FUNCTION DT_TO_SDT : SDT
VAR_INPUT
	DTI : DT;
END_VAR
VAR
	tmp : DATE;
	tdt : DWORD;
END_VAR


(*
version 1.0	18. oct 2008
programmer 	hugo
tested by	oscat

converts date_time to Structured date time (SDT)

*)

tmp := DT_TO_DATE(dti);
tdt := DT_TO_DWORD(dti) - DATE_TO_DWORD(tmp);
DT_TO_SDT.YEAR := YEAR_OF_DATE(tmp);
DT_TO_SDT.MONTH := MONTH_OF_DATE(tmp);
DT_TO_SDT.DAY := DAY_OF_MONTH(tmp);
DT_TO_SDT.WEEKDAY := DAY_OF_WEEK(tmp);
DT_TO_SDT.SECOND := DWORD_TO_INT(tdt MOD 60);
DT_TO_SDT.MINUTE := DWORD_TO_INT((tdt / 60) MOD 60);
DT_TO_SDT.HOUR := DWORD_TO_INT(tdt / 3600);

(* revision history

hm 18. oct. 2008	rev 1.0
	original version

*)

END_FUNCTION

(* stored: Version 1.1.0.1, ProductVersion 3.1.4022.7
   POU DT_TO_SDT: Id {843c4af2-790c-4155-942e-85bf545477fc}, SpecialFunc None *)
